// TIA Portal V16 export
// export: Created 2022-11-17T15:49:35.1982462Z, ExportSetting WithDefaults, DisplayName Totally Integrated Automation Portal, DisplayVersion V16 Update 6, DisplayName TIA Portal Version Control Interface, DisplayVersion V16 Update 2, DisplayName TIA Portal Openness, DisplayVersion V16 Update 6, DisplayName SINAMICS Startdrive Advanced, DisplayVersion V16 Update 5, DisplayName SINAMICS Startdrive G130, G150, S120, S150, SINAMICS MV, S210, DisplayVersion V16 Update 5, DisplayName SINAMICS Startdrive G110M, G120, G120C, G120D, G120P, G115D, DisplayVersion V16 Update 5, DisplayName STEP 7 Professional, DisplayVersion V16 Update 6, DisplayName STEP 7 Safety, DisplayVersion V16, DisplayName WinCC Advanced, DisplayVersion V16 Update 6
DATA_BLOCK "EncoderCh1-CarriageB"   // DB103
// stored: AutoNumber false, InstanceOfName CTRL_HSC, OfSystemLibElement CTRL_HSC, OfSystemLibVersion 1.0
"CTRL_HSC"
   // VAR_INPUT
   //    HSC : HW_HSC;
   //    DIR : Bool;
   //    CV : Bool;
   //    RV : Bool;
   //    PERIOD : Bool;
   //    NEW_DIR : Int;
   //    NEW_CV : DInt;
   //    NEW_RV : DInt;
   //    NEW_PERIOD : Int;
   // END_VAR
   // VAR_OUTPUT
   //    BUSY : Bool;
   //    STATUS : Word;
   // END_VAR
BEGIN
END_DATA_BLOCK
